PROGRAM main
  VAR
    RUN : BOOL;
    FAULTED : BOOL;
    START AT %IX0.0 : BOOL;
    STOP AT %IX0.1 : BOOL;
    RESET AT %IX0.2 : BOOL;
    FAULT AT %IX0.3 : BOOL;
    GREEN_LED AT %QX0.0 : BOOL;
    YELLOW_LED AT %QX0.1 : BOOL;
    RED_LED AT %QX0.2 : BOOL;
  END_VAR

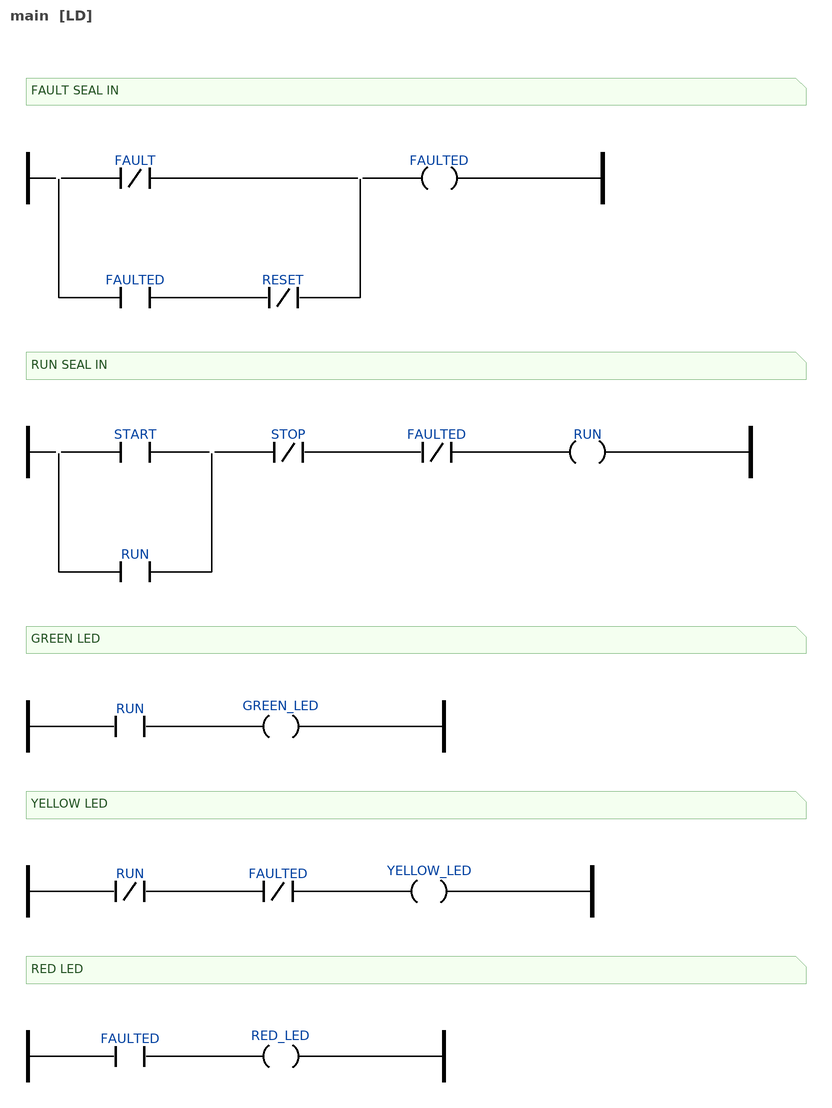
(* LD diagram, written out as Structured Text *)
(* FAULT SEAL IN *)
FAULTED := NOT FAULT OR FAULTED AND NOT RESET;
(* RUN SEAL IN *)
RUN := (START OR RUN) AND NOT STOP AND NOT FAULTED;
(* GREEN LED *)
GREEN_LED := RUN;
(* YELLOW LED *)
YELLOW_LED := NOT RUN AND NOT FAULTED;
(* RED LED *)
RED_LED := FAULTED;
END_PROGRAM
